	19206:
		F_ADSErrorCodeExt := 'Parameter incorrect. Override outside bounds, or read/write parameter type mismatch.';

	19207:
		F_ADSErrorCodeExt := 'Timeout axis function block. Position range monitoring time exceeded, target position monitoring time exceeded.';

	19208:
		F_ADSErrorCodeExt := 'The axis is in protected mode (e.g., coupled) and cannot be moved.';

	19209:
		F_ADSErrorCodeExt := 'Axis is not ready.';

	19210:
		F_ADSErrorCodeExt := 'Error during referencing.';

	19211:
		F_ADSErrorCodeExt := 'The definition of the trigger signal for function block MC_TouchProbe is incorrect..';

	19212:
		F_ADSErrorCodeExt := 'Position latch was disabled after MC_Touchprobe execute.';

	19213:
		F_ADSErrorCodeExt := 'NC status feedback timeout. An expected feedback in the axis status word has not arrived.';

	19214:
		F_ADSErrorCodeExt := 'Additional product not installed.';

	19215:
		F_ADSErrorCodeExt := 'No NC Cycle Counter Update.';

	19216:
		F_ADSErrorCodeExt := 'M-function query missing.';

	19217:
		F_ADSErrorCodeExt := 'Zero shift index is outside the range. The index of the zero shift is invalid.';

	19218:
		F_ADSErrorCodeExt := 'R-parameter index or size is invalid. This error occurs if the R-parameters are written or read but the index or size are outside the range.';

	19219:
		F_ADSErrorCodeExt := 'Index for tool description is invalid.';

	19220:
		F_ADSErrorCodeExt := 'Version of the cyclic channel interface does not match the requested function or the function block.';

	19221:
		F_ADSErrorCodeExt := 'Channel is not ready for the requested function.';

	19222:
		F_ADSErrorCodeExt := 'The requested function requires explicit activation.';

	19223:
		F_ADSErrorCodeExt := 'Axis is already in another group.';

	19224:
		F_ADSErrorCodeExt := 'Block search could not be executed successfully.';

	19225:
		F_ADSErrorCodeExt := 'This error occurs if the FB ItpBlocksearch is called with invalid parameters (e.g., E_ItpDryRunMode, E_ItpBlockSearchMode)';

	19232:
		F_ADSErrorCodeExt := 'Cannot add all axes to the interpolation group.';

	19248:
		F_ADSErrorCodeExt := 'A pointer to a data structure is invalid, e.g., Null';

	19249:
		F_ADSErrorCodeExt := 'The specification of the memory size (SIZE) for a data structure is invalid.';

	19250:
		F_ADSErrorCodeExt := 'Cam table ID is invalid.';

	19251:
		F_ADSErrorCodeExt := 'Point ID is invalid. The ID of a point (sampling point) of a motion function is less than 1.';

	19252:
		F_ADSErrorCodeExt := 'The number of points (sampling points) of a cam plate to be read or written is less than 1.';

	19253:
		F_ADSErrorCodeExt := 'The type of a cam plate does not match the definition MC_TableType.';

	19254:
		F_ADSErrorCodeExt := 'The number of rows (sampling points) of a cam table is less than 1.';

	19255:
		F_ADSErrorCodeExt := 'The number of columns of a cam table is invalid.';

	19256:
		F_ADSErrorCodeExt := 'Step size invalid. The increment for the interpolation is invalid, e.g., less than or equal to zero.';

	19264:
		F_ADSErrorCodeExt := 'The terminal used is not supported by this function block.';

	19265:
		F_ADSErrorCodeExt := 'Register read/write error. This error implies a validity error.';

	19266:
		F_ADSErrorCodeExt := 'The axis is enabled but should not be enabled for this process.';

	19267:
		F_ADSErrorCodeExt := 'Incorrect size of the compensation table. The specified table size (in bytes) does not match the actual size';

	19268:
		F_ADSErrorCodeExt := 'The minimum/maximum position in the compensation table does not match the position in the table description (ST_CompensationDesc)';

	19269:
		F_ADSErrorCodeExt := 'The requested function is not implemented in this combination';

	19270:
		F_ADSErrorCodeExt := 'Window not in the specified modulo range.';

	19271:
		F_ADSErrorCodeExt := 'Buffer overflow. The number of events has led to an overflow of the buffer and not all events could be acquired.';

	19296:
		F_ADSErrorCodeExt := 'Motion command did not become active.';

	19297:
		F_ADSErrorCodeExt := 'Motion command could not be monitored by the PLC.';

	19298:
		F_ADSErrorCodeExt := 'A buffered command was terminated with an error.';

	19299:
		F_ADSErrorCodeExt := 'A buffered command was completed but there was no feedback to indicate success or failure.';

	19300:
		F_ADSErrorCodeExt := 'The BufferMode is not supported by this command.';

	19301:
		F_ADSErrorCodeExt := 'The command number for queued commands managed by the system unexpectedly has the value 0.';

	19302:
		F_ADSErrorCodeExt := 'Function block was not called cyclically.';

	19313:
		F_ADSErrorCodeExt := 'Invalid NCI entry type. The FB FB_NciFeedTablePreparation was called with an unknown nEntryType.';

	19314:
		F_ADSErrorCodeExt := 'NCI feed table is full and the entry is therefore not accepted.';

	19315:
		F_ADSErrorCodeExt := 'Internal error.';

	19316:
		F_ADSErrorCodeExt := 'ST_NciTangentialFollowingDesc: Tangential axis is not an auxiliary axis.';

	19317:
		F_ADSErrorCodeExt := 'ST_NciTangentialFollowingDesc: nPathAxis1 or nPathAxis2 is not a path axis. It is therefore not possible to determine the plane.';

	19318:
		F_ADSErrorCodeExt := 'ST_NciTangentialFollwoingDesc: nPathAxis1 and nPathAxis2 are the same. It is therefore not possible to determine the plane.';

	19319:
		F_ADSErrorCodeExt := 'ST_NciGeoCirclePlane: Circle incorrectly parameterized';

	19320:
		F_ADSErrorCodeExt := 'Internal error during calculation of tangential following';

	19321:
		F_ADSErrorCodeExt := 'Tangential following: Monitoring of the deviation angle was activated during activation of tangential following.';

	19322:
		F_ADSErrorCodeExt := 'Not implemented';

	19323:
		F_ADSErrorCodeExt := 'Tangential following: the radius of the current arc is too small';

	19324:
		F_ADSErrorCodeExt := 'FB_NciFeedTablePreparation: pEntry is NULL';

	19325:
		F_ADSErrorCodeExt := 'FB_NciFeedTablePreparation: the specified nEntryType does not match the structure type';

	19326:
		F_ADSErrorCodeExt := 'ST_NciMFuncFast and ST_NciMFuncHsk: the requested M-function is not between 0 and 159';

	19327:
		F_ADSErrorCodeExt := 'ST_NciDynOvr: the requested value for the dynamic override is not between 0.01 and 1';

	19328:
		F_ADSErrorCodeExt := 'ST_NciVertexSmoothing: invalid parameter. This error is generated if a negative smoothing radius or an unknown smoothing type is encountered.';

	19329:
		F_ADSErrorCodeExt := 'FB_NciFeedTablePrepartion: The requested velocity is not in the valid range';

	19330:
		F_ADSErrorCodeExt := 'ST_Nci*: invalid parameter';

	19344:
		F_ADSErrorCodeExt := 'Determined drive type is not supported';

	19345:
		F_ADSErrorCodeExt := 'Direction is impermissible';

	19346:
		F_ADSErrorCodeExt := 'SwitchMode is impermissible';

	19347:
		F_ADSErrorCodeExt := 'Mode for the parameter handling is impermissible';

	19348:
		F_ADSErrorCodeExt := 'Parameterization of the torque limits is inconsistent';

	19349:
		F_ADSErrorCodeExt := 'Parameterization of the position lag limit is impermissible (<=0).';

	19350:
		F_ADSErrorCodeExt := 'Parameterization of the distance limit is impermissible (<0)';

	19351:
		F_ADSErrorCodeExt := 'An attempt was made to back up parameters again, although they have already been backed up.';

	19352:
		F_ADSErrorCodeExt := 'An attempt was made to restore parameters, although none have been backed up.';

	19359:
		F_ADSErrorCodeExt := 'The abortion of a homing has failed.';

	19360:
		F_ADSErrorCodeExt := 'KinGroup error: the kinematic group is in an error state.';

	19361:
		F_ADSErrorCodeExt := 'KinGroup timeout: timeout during call of a kinematic block';

	19376:
		F_ADSErrorCodeExt := 'The current axis position or the axis position resulting from the new position offset exceeds the valid range of values.';

	19377:
		F_ADSErrorCodeExt := 'The new position offset exceeds the valid range of values [AX5000: 2^31].';

	19378:
		F_ADSErrorCodeExt := 'The current axis position or the axis position resulting from the new position offset falls below the valid range of values.';

	19379:
		F_ADSErrorCodeExt := 'The new position offset falls below the valid range of values [AX5000: -2^31].';

	19380:
		F_ADSErrorCodeExt := 'The activated feedback and/or storage location (AX5000: P-0-0275) differ from the parameterization on the function block.';

	19381:
		F_ADSErrorCodeExt := 'Reinitialization of the actual NC position has failed, e.g., reference system = “ABSOLUTE (with single overflow)” & software end position monitoring is disabled.';

	19382:
		F_ADSErrorCodeExt := 'The command to set or delete a position offset was rejected without feedback data, e.g., if the drive controllers firmware does not support the corresponding command.';

	19383:
		F_ADSErrorCodeExt := 'The command to set or delete a position offset was rejected with feedback data. The information in the feedback data may contain further information about the cause.';

	19384:
		F_ADSErrorCodeExt := 'A firmware version >= 19 is required for the servo terminal.';

	19385:
		F_ADSErrorCodeExt := 'The modulo settings on the drive controller and NC are different.';

	19394:
		F_ADSErrorCodeExt := 'The new position offset exceeds the valid value range.';

	19395:
		F_ADSErrorCodeExt := 'I/O data are invalid or the terminal is in an error state.';

	// TF6310 TCP/IP

	// 32769 - 32773
	32769:
		F_ADSErrorCodeExt := 'No new sockets can be created (for FB_SocketListen and FB_SocketConnect)';

	32770:
		F_ADSErrorCodeExt := 'Socket handle is invalid (for FB_SocketReceive, FB_SocketAccept, FB_SocketSend etc.)';

	32771:
		F_ADSErrorCodeExt := 'TcpIp port listener already exists (returned from FB_SocketListen)';

	32772:
		F_ADSErrorCodeExt := 'Client socket is no longer connected with the server (returned from FB_SocketReceive)';

	32773:
		F_ADSErrorCodeExt := 'Error was registered in the listener socket (returned from FB_SocketAccept)';

	// Win32 Errors	
	16#8007274C:
		F_ADSErrorCodeExt := CONCAT('Win32 system error - ', 'A connection attempt failed because the connected party did not properly respond after a period of time, or the established connection failed because the connected host failed to respond.');

ELSE
	IF ErrorId >= 16#80070000 AND ErrorId <= 16#8007FFFF THEN
		CONCAT(CONCAT('Win32 system error - ', TO_STRING(ErrorId)), ', Not Found');
	ELSE
		IF ErrorId = 33056 THEN
			F_ADSErrorCodeExt := 'Invalid configuration for Object (e.g. in System Manager).';
		ELSIF ErrorId = 33057 THEN
			F_ADSErrorCodeExt := 'Invalid environment for Object (e.g. TcCom-Objects Hierarchy or missing/faulty Objects).';
		elsif ErrorId = 33058 Then
			F_ADSErrorCodeExt := 'Incompatible Driver or Object.';
		elsif ErrorId = 33060 Then
			F_ADSErrorCodeExt := 'Command execution does not terminate (e. g. MC_Reset does not signal DONE).';
		elsif ErrorId = 33072 Then
			F_ADSErrorCodeExt := 'Invalid ObjectID of Communication Target.';
		elsif ErrorId = 33073 Then
			F_ADSErrorCodeExt := 'Communication Target expects Call in different Context.';
		elsif ErrorId = 33074 Then
			F_ADSErrorCodeExt := 'Invalid State of Communication Target.';
		elsif ErrorId = 33076 Then
			F_ADSErrorCodeExt := 'Communication with Communication Target cannot be established.';
		elsif ErrorId = 33083 Then
			F_ADSErrorCodeExt := 'Transition Mode is invalid.';
		elsif ErrorId = 33084 Then
			F_ADSErrorCodeExt := 'BufferMode is invalid.';
		elsif ErrorId = 33085 Then
			F_ADSErrorCodeExt := 'Only one active Instance of Function Block per Group is allowed.';
		elsif ErrorId = 33086 Then
			F_ADSErrorCodeExt := 'Command is not allowed in current group state.';
		elsif ErrorId = 33087 Then
			F_ADSErrorCodeExt := 'Slave cannot synchronize. The slave cannot reach the SlaveSyncPosition with the given dynamics.';
		elsif ErrorId = 33088 Then
			F_ADSErrorCodeExt := 'Invalid value for one or more of the dynamic parameters (Acceleration, Deceleration, Jerk).';
		elsif ErrorId = 33089 Then
			F_ADSErrorCodeExt := 'IdentInGroup is invalid.';
		elsif ErrorId = 33090 Then
			F_ADSErrorCodeExt := 'The number of axes in the group is incompatible with the axes convention.';
		elsif ErrorId = 33091 Then
			F_ADSErrorCodeExt := 'Function Block or respective Command is not supported by Target.';
		elsif ErrorId = 33092 Then
			F_ADSErrorCodeExt := 'Command queue full. Command queue is completely filled up and cannot accept additional commands until some commands are fully processed.';
		elsif ErrorId = 33093 Then
			F_ADSErrorCodeExt := 'Mapping of Cyclic Interface between NC and PLC is missing (e.g. AXIS_REF, AXES_GROUP_REF, ...).';
		elsif ErrorId = 33094 Then
			F_ADSErrorCodeExt := 'Invalid Velocity Value. The velocity was not set or the entered value is invalid.';
		elsif ErrorId = 33095 Then
			F_ADSErrorCodeExt := 'Invalid Coordinate Dimension. The dimension of the set coordinate interpretation does not meet the requirements.';
		elsif ErrorId = 33096 Then
			F_ADSErrorCodeExt := 'Invalid Input Value.';
		elsif ErrorId = 33097 Then
			F_ADSErrorCodeExt := 'Unsupported Dynamics for selected Group Kernel.';
		elsif ErrorId = 33098 Then
			F_ADSErrorCodeExt := 'The programmed position dimension incompatible with the axes convention.';
		elsif ErrorId = 33099 Then
			F_ADSErrorCodeExt := 'Path buffer is invalid. E.g. because provided buffer has invalid address or is not big enough.';
		elsif ErrorId = 33100 Then
			F_ADSErrorCodeExt := 'Path does not contain any element.';
		elsif ErrorId = 33101 Then
			F_ADSErrorCodeExt := 'Provided Path buffer is too small to store more Path Elements.';
		elsif ErrorId = 33102 Then
			F_ADSErrorCodeExt := 'Dimension or at least one Value of Transition Parameters is invalid.';
		elsif ErrorId = 33103 Then
			F_ADSErrorCodeExt := 'Invalid or Incomplete Input Array.';
		elsif ErrorId = 33104 Then
			F_ADSErrorCodeExt := 'Path length is zero.';
		elsif ErrorId = 33105 Then
			F_ADSErrorCodeExt := 'Command is not allowed in current axis state.';
		elsif ErrorId = 33106 Then
			F_ADSErrorCodeExt := 'TwinCAT System is shutting down and cannot complete request.';
		elsif ErrorId = 33107 Then
			F_ADSErrorCodeExt := 'Configured axes convention and configured axes do not match.';
		elsif ErrorId = 33108 Then
			F_ADSErrorCodeExt := 'Invalid Number of ACS Axes. The number of ACS input axes does not match the number of ACS input axes expected by the kinematic transformation.';
		elsif ErrorId = 33109 Then
			F_ADSErrorCodeExt := 'Invalid Number of MCS Data. The number of MCS input data does not match the number expected by the kinematic transformation.';
		elsif ErrorId = 33110 Then
			F_ADSErrorCodeExt := 'Invalid Value Set for Kinematic Parameters. The numeric value set for the parameter does not reside within the respective definition range.';
		elsif ErrorId = 33112 Then
			F_ADSErrorCodeExt := 'The Given ACS Values Cannot be Reached. The given ACS values result in an invalid machine configuration.';
		elsif ErrorId = 33113 Then
			F_ADSErrorCodeExt := 'The Set Target Positions Cannot be Reached. The set target positions reside outside the admissible working space.';
		elsif ErrorId = 33117 Then
			F_ADSErrorCodeExt := 'Discontinuity in ACS axes detected.';
		elsif ErrorId = 33120 Then
			F_ADSErrorCodeExt := 'Circle Specification in Path is invalid. The specification of a circle segment in the programmed interpolated path (e.g. via MC_MovePath) has an invalid or ambiguous description. Probably its center cannot be determined reliably.';
		elsif ErrorId = 33121 Then
			F_ADSErrorCodeExt := 'Maximum stream lines reached. The maximum number of stream lines is limited. Please refer to function block documentation for details.';
		elsif ErrorId = 33123 Then
			F_ADSErrorCodeExt := 'Invalid First Segment. The corresponding element can only be analyzed with a well-defined start point.';
		elsif ErrorId = 33124 Then
			F_ADSErrorCodeExt := 'Invalid auxiliary point. The auxiliary point is not well-defined.';
		elsif ErrorId = 33126 Then
			F_ADSErrorCodeExt := 'Invalid parameter for GapControlMode. Invalid parameter for GapControlMode, most likely in combination with the group parameter GapControlDirection.';
		elsif ErrorId = 33127 Then
			F_ADSErrorCodeExt := 'Group got unsupported Axis Event (e.g. State Change). Group got unsupported Axis Event (e.g. State Change e.g. triggered by a Single Axis Reset).';
		elsif ErrorId = 33128 Then
			F_ADSErrorCodeExt := 'Unsupported Compensation Type. The compensation type was either not set or is not supported by the addressed object.';
		elsif ErrorId = 33129 Then
			F_ADSErrorCodeExt := 'Master axis does not exist or cannot be used.';
		elsif ErrorId = 33130 Then
			F_ADSErrorCodeExt := 'Invalid or Missing Tracking Transformation. This error occurs at MC_TrackConveyorBelt if at the CoordTransform input an invalid object ID is used or the object ID points to an object that is not supported as coordinate transformation.';
		elsif ErrorId = 33131 Then
			F_ADSErrorCodeExt := 'Position is not on Track. Either Track cannot be activated because Actual Position is not on Track, or Target Position is not on Active Track or TrackPart.';
		elsif ErrorId = 33132 Then
			F_ADSErrorCodeExt := 'Axis does not have an activated track.';
		elsif ErrorId = 33133 Then
			F_ADSErrorCodeExt := 'Invalid Compensation ObjectId. An Object with this ObjectId does not exist or it is not of the right type (has to be a compensation).';
		elsif ErrorId = 33134 Then
			F_ADSErrorCodeExt := 'Axis is in error because axis was not in Target when InTargetAlarm Timer expired.';
		elsif ErrorId = 33135 Then
			F_ADSErrorCodeExt := 'Coupling would cause a cyclic dependency of axis (e.g. via MC_GearInPos).';
		elsif ErrorId = 33136 Then
			F_ADSErrorCodeExt := 'Axis was not added to an axes group, the command is not valid.';
		elsif ErrorId = 33151 Then
			F_ADSErrorCodeExt := 'Drive has invalid State.';
		elsif ErrorId = 33153 Then
			F_ADSErrorCodeExt := 'Parameter for gap control are invalid with the current configuration. Function block with gap control was issued to an axis that is not in a CA group.';
		elsif ErrorId = 33154 Then
			F_ADSErrorCodeExt := 'Software position limit violation. Software position limits of at least one axis have been or would have been violated by a command.';
		elsif ErrorId = 33155 Then
			F_ADSErrorCodeExt := 'Target position is not reachable. There is no path available to the target position or target position is unreachable in general.';
		elsif ErrorId = 33157 Then
			F_ADSErrorCodeExt := 'The mover or one of its relevant coordinates is busy. Either the whole mover or at least of its coordinates relevant to the command are busy.';
		elsif ErrorId = 33158 Then
			F_ADSErrorCodeExt := 'A collision has occurred or would occur. Either a collision has occurred or would occur if the command was executed.';
		elsif ErrorId = 33159 Then
			F_ADSErrorCodeExt := 'Invalid Track Specification. The geometric extension of this track is incompatible with the already existing geometry of this or the other tracks.';
		elsif ErrorId = 33160 Then
			F_ADSErrorCodeExt := 'Command not allowed in track state.';
		elsif ErrorId = 33161 Then
			F_ADSErrorCodeExt := 'Invalid Reference passed to Function Block. An invalid reference (or pointer) was used in a function block call. This can happen if a reference type is used before it was initialized.';
		elsif ErrorId = 33162 Then
			F_ADSErrorCodeExt := 'Path is locked against modifications. The path was locked to further changes. However, it might be resettable.';
		ELSIF ErrorId = 33164 THEN
			F_ADSErrorCodeExt := 'Position out of modulo range. Position must be larger or equal to zero and less or equal to the modulo factor when using modulo positioning.';
		elsif ErrorId = 33165 Then
			F_ADSErrorCodeExt := 'The specified value AdditionalTurns at the Options input is not allowed. The parameter AdditionalTurns must be zero for the specified value of the parameter Direction.';
		elsif ErrorId = 33166 Then
			F_ADSErrorCodeExt := 'Master/Slave sync position incompatible with sync direction. The given sync positions require the slave moving in a direction which is not allowed while in synchronization phase.';
		ELSE
			F_ADSErrorCodeExt := CONCAT('ADS Error Code - ', TO_STRING(ErrorId));
		END_IF
	END_IF
END_CASE

END_FUNCTION

// FunctionBlocks/FB_Component_NciParameterBase
FUNCTION_BLOCK FB_Component_NciParameterBase EXTENDS FB_ComponentBase
VAR
	ipChannel : I_NciChannel;

	// Alarms
	ComponentNciParameterAlarms : ARRAY[1..COMPONENT_NCI_PARAMETER_ALARM_COUNT] OF FB_TcAlarm;
END_VAR

VAR CONSTANT
	COMPONENT_NCI_PARAMETER_ALARM_COUNT : UDINT := 2;
END_VAR

//! @summary Clears error flags and error IDs for this component
METHOD PUBLIC Reset : BOOL
F_ClearAllEventsInClass(ComponentNciParameterAlarms);
_Error	 := FALSE;
_ErrorId := 0;
Reset	 := SUPER^.Reset();
END_METHOD

//! @summary This method serves as the entry point for all underlying FB logic
METHOD PUBLIC CyclicLogic

//! @description This method should be called cyclically by descendant function blocks by invoking <c>SUPER^.CyclicLogic()</c>.  Alternatively, the contents of this method could be reimplemented entirely in which case a call to this method would not be necessary.
IF NOT _InitComplete THEN
	_InitComplete := Initialize();
	RETURN;
END_IF

// Call Super
SUPER^.CyclicLogic();
_CurrentAlarmSeverity := F_GetMaxSeverityRaised(Alarms := ComponentNciParameterAlarms, CurrentSeverity := _CurrentAlarmSeverity);
END_METHOD

//! @summary Initializes event function blocks using this components's name
METHOD PROTECTED CreateEvents

//! @description This method is called by <c>Initialize()</c> as required
SUPER^.CreateEvents();
F_CreateAllEventsInClass(Alarms		:= ComponentNciParameterAlarms,
						 ClassSize	:= SIZEOF(TC_EVENTS.NciParameterAlarms),
						 pInitEvent := ADR(TC_EVENTS.NciParameterAlarms.InitReferenceEvent),
						 Prefix		:= _Name);
END_METHOD

PROPERTY Channel : I_NciChannel
SET
ipChannel := Channel;
END_SET
END_PROPERTY

//! @summary Basic component initialization logic
METHOD PROTECTED Initialize : BOOL;

//! @description This method is called by <c>CyclicLogic()</c> as required
IF ipChannel = 0 THEN
	TRACE('Nci Channel not assigned!');
	_Error	 := TRUE;
	_ErrorId := 1;
	RETURN;
END_IF

Initialize := Super^.Initialize();
END_METHOD

END_FUNCTION_BLOCK

// FunctionBlocks/FB_Component_NciReadWriteRParameter
FUNCTION_BLOCK FB_Component_NciReadWriteRParameter EXTENDS FB_Component_NciParameterBase
VAR
	// Write R-Parameter
	WriteRParamsEx : ItpWriteRParamsEx;

	// Read R-Parameter
	ReadRParamsEx : ItpReadRParamsEx;
END_VAR

//! @summary Clears error flags and error IDs for this component
METHOD PUBLIC Reset : BOOL
F_ClearAllEventsInClass(ComponentNciParameterAlarms);
_Error	 := FALSE;
_ErrorId := 0;
Reset	 := SUPER^.Reset();
END_METHOD

//! @summary This method serves as the entry point for all underlying FB logic
METHOD PUBLIC CyclicLogic

//! @description This method should be called cyclically by descendant function blocks by invoking <c>SUPER^.CyclicLogic()</c>.  Alternatively, the contents of this method could be reimplemented entirely in which case a call to this method would not be necessary.
IF NOT _InitComplete THEN
	_InitComplete := Initialize();
	RETURN;
END_IF

// Read
ReadRParamsEx(sNciToPlc := ipChannel.Channel.NcToPLC, tTimeOut := T#1S);
IF ReadRParamsEx.bErr AND ReadRParamsEx.bExecute THEN
	_Error	 := TRUE;
	_ErrorId := ReadRParamsEx.nErrId;
END_IF

IF NOT ReadRParamsEx.bBusy THEN
	ReadRParamsEx.bExecute := FALSE;
END_IF

// Write
WriteRParamsEx(sNciToPlc := ipChannel.Channel.NcToPLC, tTimeOut := T#1S);
IF WriteRParamsEx.bErr AND WriteRParamsEx.bExecute THEN
	_Error	 := TRUE;
	_ErrorId := WriteRParamsEx.nErrId;
END_IF

IF NOT WriteRParamsEx.bBusy THEN
	WriteRParamsEx.bExecute := FALSE;
END_IF

//
_Busy := ReadRParamsEx.bBusy OR WriteRParamsEx.bBusy;

// Call Super
SUPER^.CyclicLogic();
END_METHOD

//! Provides basic error detection and event handling for this component
METHOD PROTECTED Monitoring
VAR_INST
	RTrigError	: R_TRIG; // Error active - Error Bit remains On in NCI Fbs until new command is issued
	TempMessage : STRING;
END_VAR

(*! @descriptionThis method is called cyclically by <c>CyclicLogic()</c>*)
SUPER^.Monitoring();
RTrigError(CLK := _Error);
IF RTrigError.Q THEN
	IF ReadRParamsEx.bErr THEN
		TempMessage := 'Read R-Parameter';
	END_IF

	IF WriteRParamsEx.bErr THEN
		TempMessage := 'Write R-Parameter';
	END_IF

	// 
	IF NOT ComponentNciParameterAlarms[E_NciParameterAlarms.ParameterError].bRaised THEN
		RaiseAlarmWithStrings(ComponentNciParameterAlarms[E_NciParameterAlarms.ParameterError], TempMessage, F_ADSErrorCodeExt(_ErrorId));
	END_IF
END_IF
END_METHOD

METHOD PUBLIC Read : BOOL
VAR_INPUT
	RParameter		: ANY;			// LREAL or Array of Lreal
	StartRParameter : UINT(0..999); // R Parameter to start reading, lenght of RParameter type is read
END_VAR

VAR CONSTANT
	SIZE_OF_LREAL	: UINT := 8;
	MAX_R_PARAMETER : UINT := 1000;
END_VAR
IF RParameter.diSize < SIZE_OF_LREAL THEN
	TRACE('RParameter Pointer is empty!');
	RETURN;
END_IF

IF RParameter.TypeClass <> __SYSTEM.TYPE_CLASS.TYPE_ARRAY AND RParameter.TypeClass <> __SYSTEM.TYPE_CLASS.TYPE_LREAL THEN
	TRACE('RParameter Datatype not LREAL or ARRAY of LREAL!');
	RETURN;
END_IF

IF (StartRParameter + (RParameter.diSize / SIZE_OF_LREAL)) > MAX_R_PARAMETER THEN
	TRACE('StartRParameter + Size of RParameter is larger than 1000 R Parameters!');
	RETURN;
END_IF

IF _Error OR _Busy THEN
	RETURN;
END_IF

ReadRParamsEx.bExecute := TRUE;
ReadRParamsEx.pAddr	   := RParameter.pValue;
ReadRParamsEx.nIndex   := StartRParameter;
ReadRParamsEx.nCount   := (RParameter.diSize / SIZE_OF_LREAL);
Read				   := TRUE;
END_METHOD

METHOD PUBLIC Write : BOOL
VAR_INPUT
	RParameter		: ANY;			// LREAL or Array of Lreal
	StartRParameter : UINT(0..999); // R Parameter to write, lenght of RParameter type is written
END_VAR

VAR CONSTANT
	SIZE_OF_LREAL	: UINT := 8;
	MAX_R_PARAMETER : UINT := 1000;
END_VAR
IF RParameter.diSize < SIZE_OF_LREAL THEN
	TRACE('RParameter Pointer is empty!');
	RETURN;
END_IF

IF RParameter.TypeClass <> __SYSTEM.TYPE_CLASS.TYPE_ARRAY AND RParameter.TypeClass <> __SYSTEM.TYPE_CLASS.TYPE_LREAL THEN
	TRACE('RParameter Datatype not LREAL or ARRAY of LREAL!');
	RETURN;
END_IF

IF (StartRParameter + (RParameter.diSize / SIZE_OF_LREAL)) > MAX_R_PARAMETER THEN
	TRACE('StartRParameter + Size of RParameter is larger than 1000 R Parameters!');
	RETURN;
END_IF

IF _Error OR _Busy THEN
	RETURN;
END_IF

WriteRParamsEx.bExecute := TRUE;
WriteRParamsEx.pAddr	:= RParameter.pValue;
WriteRParamsEx.nIndex	:= StartRParameter;
WriteRParamsEx.nCount	:= (RParameter.diSize / SIZE_OF_LREAL);
Write					:= TRUE;
END_METHOD

END_FUNCTION_BLOCK

// Project Information/F_GetCompany
// This function has been automatically generated from the project information.
{attribute 'signature_flag' := '1073741824'}
{attribute 'TcGenerated'}
{attribute 'no-analysis'}
FUNCTION F_GetCompany : WSTRING
VAR_INPUT
	
END_VAR

F_GetCompany := "Beckhoff Automation LLC";

END_FUNCTION

// Project Information/F_GetTitle
// This function has been automatically generated from the project information.
{attribute 'signature_flag' := '1073741824'}
{attribute 'TcGenerated'}
{attribute 'no-analysis'}
FUNCTION F_GetTitle : WSTRING
VAR_INPUT
	
END_VAR

F_GetTitle := "SPT NCI";

END_FUNCTION

// Project Information/F_GetVersion
// This function has been automatically generated from the project information.
{attribute 'signature_flag' := '1073741824'}
{attribute 'TcGenerated'}
{attribute 'no-analysis'}
FUNCTION F_GetVersion : ST_LibVersion
VAR_INPUT
	
END_VAR

F_GetVersion.iMajor := 3;
F_GetVersion.iMinor := 2;
F_GetVersion.iBuild := 2;
F_GetVersion.iRevision := 0;
F_GetVersion.sVersion := '3.2.2';
F_GetVersion.nFlags := 1;

END_FUNCTION
